// TIA Portal project "S7-1500 için MOVE Komutu" (V18)

(* hardware
DEVICE "S7-1500/ET200MP station_1"  S7-1500 station
   slot 0: "Rail_0"  Rack  6ES7 590-1***0-0AA0
   slot 1: "PLC_1"  CPU 1512C-1 PN  6ES7 512-1CK00-0AB0  V2.8
      slot 3: "CPU display_1"  6ES7591-1AA00-0AA0
      slot 32768: "PROFINET interface_1"  X1
         slot 32769: "Port_1"  X1 P1
         slot 32770: "Port_2"  X1 P2
      slot 34817: "Virtual CP interface port_1"  Virtual CP interface port  Virtual CP interface port
*)

// ===== PLC "PLC_1"  CPU 1512C-1 PN =====

VAR_GLOBAL   // PLC tag table "Default tag table"
   "Tag_1" AT %I0.0 : Bool;
   "Tag_2" AT %MW10 : Int;
   "Tag_3" AT %Q0.0 : Bool;
   "Tag_4" AT %I0.1 : Bool;
   "Tag_5" AT %Q0.1 : Bool;
   "Tag_6" AT %MW11 : Int;
   "Tag_7" AT %MW12 : Int;
   "Tag_8" AT %MW13 : Int;
   "Tag_9" AT %MW14 : Int;
END_VAR

ORGANIZATION_BLOCK "Main"   // OB1, LAD, ProgramCycle
TITLE = "Main Program Sweep (Cycle)"
{ S7_Optimized_Access := 'TRUE' }
VERSION : 0.1
   VAR_INPUT
      Initial_Call : Bool;   // Initial call of this OB
      Remanence : Bool;   // =True, if remanent data are available
   END_VAR
BEGIN

REGION Network 1: I0.0 basınca MW10 adresine 3 değeri girilecek. Aktarma gerçekleşince Q0.0 çıkışı çalışır.
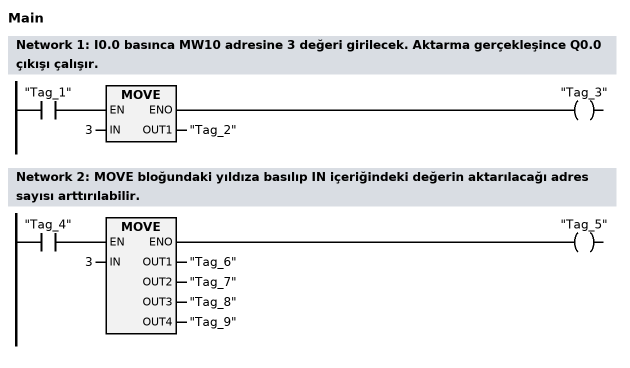
   RUNG wire#powerrail
      Contact( "Tag_1" )
      Move(in := 3, out1 => "Tag_2")
      Coil( "Tag_3" )
   END_RUNG
   // the same network as SCL:
   IF "Tag_1" THEN "Tag_2" := 3; END_IF;
   "Tag_3" := "Tag_1";
END_REGION

REGION Network 2: MOVE bloğundaki yıldıza basılıp IN içeriğindeki değerin aktarılacağı adres sayısı arttırılabilir.
   RUNG wire#powerrail
      Contact( "Tag_4" )
      Move(in := 3, out1 => "Tag_6", out2 => "Tag_7", out3 => "Tag_8", out4 => "Tag_9")
      Coil( "Tag_5" )
   END_RUNG
   // the same network as SCL:
   IF "Tag_4" THEN
       "Tag_6" := 3;
       "Tag_7" := 3;
       "Tag_8" := 3;
       "Tag_9" := 3;
   END_IF;
   "Tag_5" := "Tag_4";
END_REGION
END_ORGANIZATION_BLOCK